// TwinCAT 3 PLC project Main_Lube_oil_Temperature_Simulation
// ProgramVersion: 3.1.4024.0
// libraries:
//   Tc2_Standard, * (Beckhoff Automation GmbH)
//   Tc2_System, * (Beckhoff Automation GmbH)
//   Tc3_Module, * (Beckhoff Automation GmbH)
//   Tc2_ControllerToolbox,3.4.3.0,Beckhoff Automation GmbH
// project tree:
//   GVLs/ MainLubeOil_Parameters.TcGVL, Simulation_Parameters.TcGVL
//   / PlcTask.TcTTO
//   POUs/ FB_RampGeneration.TcPOU, FB_ReservoirVolume.TcPOU, FB_PumpFlow.TcPOU, FB_TemperatureAfterGearbox.TcPOU, FB_TemperatureAfterPump.TcPOU, FB_TemperatureAfterHeatExchanger.TcPOU, F_Scale.TcPOU, MAIN.TcPOU, f_CalculateDeltaT.TcPOU, f_deltaT_AfterMixingTwoFluids.TcPOU, FB_ReservoirTemperature.TcPOU, FB_ReservoirHeaterIsOn.TcPOU, f_ReservoirConvectionHeat.TcPOU
// real-time tasks:
//   TASK PlcTask: cycle T#10ms, priority 20, ADS port 350

CONFIGURATION Main_Lube_oil_Temperature_Simulation
    RESOURCE PLC ON TwinCAT3
        TASK PlcTask(INTERVAL := T#10ms, PRIORITY := 20);
        PROGRAM MAIN WITH PlcTask : MAIN;
    END_RESOURCE
END_CONFIGURATION

// ---- GVLs/MainLubeOil_Parameters.TcGVL
{attribute 'qualified_only'}
VAR_GLOBAL CONSTANT
	MainLubeOilReservoirVolume : REAL := 900 ; //Liters
	MainLubeOilTotalPipeVolume: REAL := 150 ; //Liters
	
	MainLubeOilReservoirHeaterPower : REAL := 5000 ; //Watt
	MainLubeOilReservoirHeaterSPon :  REAL := 40 ; // Celcius
	MainLubeOilReservoirHeaterSPoff :  REAL := 50 ; // Celcius
	
	MainLubeOilHeatExchangerPower :  REAL := 50000 ; //Watt
	MainLubeOilHeatExchangerValveClosedTemp :  REAL := 40 ; //Celcius, Valve 0% no cooling
	MainLubeOilHeatExchangerValveOpenTemp :  REAL := 80 ; //Celcius Valve 100% max cooling
	
	
	MainLubeOilPumpPower  :  REAL := 5000 ; //Watt
	MainLubeOilPumpEfficiency :  REAL := 0.95 ; // % formatted as a decimal
	
	MainLubeOilGearboxHeat :  REAL := 5000000 ; // Watt
	MainLubeOilGearboxEfficiency :  REAL := 0.993 ; // % formatted as a deimal number
	MainLubeOilGearboxStandardHeat :  REAL := 1000 ; // Watt
	
END_VAR

// ---- GVLs/Simulation_Parameters.TcGVL
{attribute 'qualified_only'}
VAR_GLOBAL CONSTANT
	OilDensity : REAL := 865 ; // g/L
	SpecificHeatCapacityOil : REAL := 2 ; // j/(g C)
	
	AmbientTemperature : REAL := 15 ; //Celcius
	GravityOilFlow : REAL := 1 ; // L/s
	CycleTime : REAL := 0.010 ; // s , 10 ms

END_VAR
VAR_GLOBAL
	TimeConstantReservoir : REAL := 0.1 ;
	TimeConstantPump : REAL := 0.0001 ;
	TimeConstantHeatExchanger : REAL := 0.0001 ;
	TimeConstantGearbox : REAL := 0.0001 ;
END_VAR

// ---- POUs/MAIN.TcPOU
PROGRAM MAIN

VAR
	fb_MainLubeOilReservoirTemperature : FB_ReservoirTemperature ;
	fb_MainLubeOilReservoirHeaterIsOn : FB_ReservoirHeaterIsOn ;
	fb_MainLubeOilTemperatureAfterPump : FB_TemperatureAfterPump ;
	fb_MainLubeOilTemperatureAfterHeatExchanger : FB_TemperatureAfterHeatExchanger ;
	fb_MainLubeOilTemperatureAfterGearbox : FB_TemperatureAfterGearbox ;
	fb_MainLubeOilReservoirVolume : FB_ReservoirVolume ;
	fb_MainLubeOilPumpFlow : FB_PumpFlow ;
	
	MainLubeOilReservoirTemperature : REAL := simulation_parameters.AmbientTemperature; // Celcius
	MainLubeOilTemperatureAfterPump : REAL := simulation_parameters.AmbientTemperature ; // Celcius
	MainLubeOilTemperatureAfterHeatExchanger : REAL := simulation_parameters.AmbientTemperature ; // Celcius
	MainLubeOilTemperatureAfterGearbox : REAL :=simulation_parameters.AmbientTemperature ; // Celcius

	MainLubeOilReservoirVolume : REAL := MainLubeOil_Parameters.MainLubeOilReservoirVolume; // L
	MainLubeOilPumpFlow  :  REAL := 0 ; // L/s
	MainLubeOilCurrentPipeVolume : REAL := 0 ; //L

	BoolSimulationTesting : BOOL := FALSE ;
	MainLubeOilReservoirHeaterIsOn : BOOL ;
	MainLubeOilPumpOneOn : BOOL := FALSE ;
	MainLubeOilPumpTwoOn : BOOL := FALSE ;
END_VAR

fb_MainLubeOilReservoirVolume(	ReservoirVolume := MainLubeOilReservoirVolume,
								ReservoirStartVolume := MainLubeOil_Parameters.MainLubeOilReservoirVolume,
								TotalPipeVolume := MainLubeOil_Parameters.MainLubeOilTotalPipeVolume,
								PumpFlow := MainLubeOilPumpFlow);

fb_MainLubeOilPumpFlow(	PumpOneOn := MainLubeOilPumpOneOn, 
						PumpTwoOn := MainLubeOilPumpTwoOn) ;
	
fb_MainLubeOilReservoirTemperature(	ReservoirVolume := MainLubeOilReservoirVolume,
									ReservoirHeaterIsOn := MainLubeOilReservoirHeaterIsOn,
									TotalPipeVolume := MainLubeOil_Parameters.MainLubeOilTotalPipeVolume,
									CurrentPipeVolume := MainLubeOilCurrentPipeVolume,
									TemperatureAfterGearbox := MainLubeOilTemperatureAfterGearbox);

									
fb_MainLubeOilReservoirHeaterIsOn(ReservoirTemperature := MainLubeOilReservoirTemperature,
								ReservoirHeaterIsOn := MainLubeOilReservoirHeaterIsOn,
								ReservoirHeaterSPon := MainLubeOil_Parameters.MainLubeOilReservoirHeaterSPon,
								ReservoirHeaterSPoff := MainLubeOil_Parameters.MainLubeOilReservoirHeaterSPoff,
								BoolSimulationTesting := BoolSimulationTesting);
								
fb_MainLubeOilTemperatureAfterPump(	TemperatureBeforePump := MainLubeOilReservoirTemperature, 
									PumpPower := MainLubeOil_Parameters.MainLubeOilPumpPower,
									PumpFlow := MainLubeOilPumpFlow,
									Density := simulation_parameters.OilDensity,
									SpecificHeatCapacity := simulation_parameters.SpecificHeatCapacityOil,
									PumpEfficiency := MainLubeOil_Parameters.MainLubeOilPumpEfficiency)	;				

fb_MainLubeOilTemperatureAfterHeatExchanger(TemperatureBeforeHeatExchanger:= MainLubeOilTemperatureAfterPump,
											HeatExchangerPower := MainLubeOil_Parameters.MainLubeOilHeatExchangerPower ,
											PumpFlow := MainLubeOilPumpFlow,
											Density := Simulation_Parameters.OilDensity,
											SpecificHeatCapacity := Simulation_Parameters.SpecificHeatCapacityOil,
											Heatexchangervalveclosedtemp :=MainLubeOil_Parameters.MainLubeOilHeatExchangerValveClosedTemp ,
											HeatExchangerValveOpenTemp := MainLubeOil_Parameters.MainLubeOilHeatExchangerValveOpenTemp,
											TotalPipeVolume := MainLubeOil_Parameters.MainLubeOilTotalPipeVolume,
											CurrentPipeVolume := MainLubeOilCurrentPipeVolume,
											BoolSimulationTesting := BoolSimulationTesting);

fb_MainLubeOilTemperatureAfterGearbox(	TemperatureBeforeGearbox:= MainLubeOilTemperatureAfterHeatexchanger,
										PumpFlow := MainLubeOilPumpFlow,
										Density := Simulation_Parameters.OilDensity,
										SpecificHeatCapacity := Simulation_Parameters.SpecificHeatCapacityOil,
										GearboxEfficiency := MainLubeOil_Parameters.MainLubeOilGearboxEfficiency,
										Gearboxheat := MainLubeOil_Parameters.MainLubeOilGearboxHeat,
										GearboxStandardHeat := MainLubeOil_Parameters.MainLubeOilGearboxStandardHeat,
										TotalPipeVolume := MainLubeOil_Parameters.MainLubeOilTotalPipeVolume,
										CurrentPipeVolume := MainLubeOilCurrentPipeVolume,
										BoolSimulationTesting := BoolSimulationTesting);								
								
MainLubeOilReservoirTemperature := fb_MainLubeOilReservoirTemperature.ReservoirTemperature ;
MainLubeOilReservoirHeaterIsOn := fb_MainLubeOilReservoirHeaterIsOn.ReservoirHeaterIsOn ;
MainLubeOilTemperatureAfterPump := fb_MainLubeOilTemperatureAfterPump.TemperatureAfterPump ;
MainLubeOilTemperatureAfterHeatExchanger := fb_MainLubeOilTemperatureAfterHeatExchanger.TemperatureAfterHeatexchanger ;
MainLubeOilTemperatureAfterGearbox := fb_MainLubeOilTemperatureAfterGearbox.TemperatureAfterGearbox ;
MainLubeOilReservoirVolume := fb_MainLubeOilReservoirVolume.ReservoirVolume ;
MainLubeOilCurrentPipeVolume := fb_MainLubeOilReservoirVolume.CurrentPipeVolume ;
MainLubeOilPumpFlow := fb_MainLubeOilPumpFlow.PumpFlow ;

END_PROGRAM

// ---- POUs/FB_ReservoirTemperature.TcPOU
FUNCTION_BLOCK FB_ReservoirTemperature
VAR_INPUT
	ReservoirVolume : REAL ; // L
	ReservoirHeaterIsOn : BOOL ;
	TotalPipeVolume : REAL ; // L
	CurrentPipeVolume : REAL ; // L
	TemperatureAfterGearbox : REAL ; //Celcius
END_VAR
VAR_OUTPUT
	ReservoirTemperature : REAL := Simulation_Parameters.AmbientTemperature ; //Celcius
END_VAR
VAR
	deltaTHeater : REAL := 0; // Celcius
	deltaTMixingGearboxReturn : REAL :=0 ; // Celcius
	
	ReservoirTemperatureNonFiltered : REAL := Simulation_Parameters.AmbientTemperature; // Celcius
	ReservoirConvectionHeat : REAL := 0 ; // Watt
	deltaTConvection : REAL := 0; // Celcius
	AmbientTemperature : REAL := Simulation_Parameters.AmbientTemperature; // Celcius
END_VAR

IF CurrentPipeVolume < (TotalPipeVolume) THEN
	deltaTMixingGearboxReturn := 0 ;
ELSE
	deltaTMixingGearboxReturn := f_deltaT_AfterMixingTwoFluids(	Mass1 := main.fb_MainLubeOilTemperatureAfterGearbox.PumpFlow,
																						SpecificHeatCapacity1 := simulation_parameters.SpecificHeatCapacityOil,
																						Temperature1 := TemperatureAfterGearbox,
																						Mass2 := ReservoirVolume,
																						SpecificHeatCapacity2 := simulation_parameters.SpecificHeatCapacityOil,
																						Temperature2 := ReservoirTemperature);
END_IF

	

IF ReservoirHeaterIsOn THEN
	deltaTHeater := f_CalculateDeltaT(	SpecificHeatCapacity := simulation_parameters.SpecificHeatCapacityOil,
										Density := Simulation_Parameters.OilDensity,
										Mass := ReservoirVolume,
										PowerInput := MainLubeoil_parameters.MainLubeOilReservoirHeaterPower);
ELSIF NOT ReservoirHeaterIsOn  THEN
	deltaTHeater := 0;
END_IF

ReservoirConvectionHeat := f_ReservoirConvectionHeat(ReservoirTemperature := ReservoirTemperature,
														AmbientTemperature := AmbientTemperature) ;
deltaTConvection := f_CalculateDeltaT (	SpecificHeatCapacity := simulation_parameters.SpecificHeatCapacityOil,
										Density := Simulation_Parameters.OilDensity,
										Mass := ReservoirVolume,
										PowerInput := ReservoirConvectionHeat);
										
ReservoirTemperatureNonFiltered := ReservoirTemperature + deltaTHeater + deltaTMixingGearboxReturn - deltaTConvection;
ReservoirTemperature := (1-simulation_parameters.TimeConstantReservoir)*ReservoirTemperature + simulation_parameters.TimeConstantReservoir*ReservoirTemperatureNonFiltered ;

END_FUNCTION_BLOCK

// ---- POUs/f_deltaT_AfterMixingTwoFluids.TcPOU
FUNCTION f_deltaT_AfterMixingTwoFluids : REAL
VAR_INPUT
	Mass1 : REAL ; // g
	SpecificHeatCapacity1 : REAL ; //  j/(g C), 
	Temperature1 : REAL ; // Celcius
	
	Mass2 : REAL ; // g
	SpecificHeatCapacity2 : REAL ; //  j/(g C), 
	Temperature2 : REAL ; // Celcius
END_VAR

f_deltaT_AfterMixingTwoFluids := ((Mass1 * SpecificHeatCapacity1 * Temperature1)+(Mass2 * SpecificHeatCapacity2 * Temperature2))/((Mass1 * SpecificHeatCapacity1 )+(Mass2 * SpecificHeatCapacity2 )) - Temperature2;

END_FUNCTION

// ---- POUs/f_CalculateDeltaT.TcPOU
FUNCTION f_CalculateDeltaT : REAL

VAR_INPUT
	PowerInput : REAL ; // Watts
	Density : REAL ; // g/L
	SpecificHeatCapacity : REAL ; // j/(g C)
	Mass : REAL; // g
END_VAR

IF Density =0 OR SpecificHeatCapacity =0 OR Mass =0 THEN 
	f_CalculateDeltaT := 0 ; 
ELSIF Mass < 0.3 THEN  //Filter to prevent large spikes when dividing by very small mass numbers.
	f_CalculateDeltaT := 0 ; 
ELSE
	f_CalculateDeltaT := PowerInput / (Density * SpecificHeatCapacity * Mass);
END_IF

END_FUNCTION

// ---- POUs/f_ReservoirConvectionHeat.TcPOU
FUNCTION f_ReservoirConvectionHeat : REAL
VAR_INPUT
	ReservoirTemperature : REAL ; // Celcius
	AmbientTemperature : REAL ; // Celcius
END_VAR
VAR_OUTPUT
	ReservoirConvectionHeat: REAL ; // Watt
END_VAR
VAR
	ConvectiveHeatTransferCoeff : REAL := 10 ; // Watt/(m2 K)
	ReservoirSurfaceArea : REAL :=6 ; // m2
END_VAR

f_ReservoirConvectionHeat := ConvectiveHeatTransferCoeff * ReservoirSurfaceArea * (ReservoirTemperature - AmbientTemperature);

END_FUNCTION

// ---- POUs/FB_ReservoirHeaterIsOn.TcPOU
FUNCTION_BLOCK FB_ReservoirHeaterIsOn
VAR_INPUT
	ReservoirTemperature : REAL ; // Celcius
	ReservoirHeaterIsOn : BOOL ; 
	ReservoirHeaterSPon : REAL ; // Celcius
	ReservoirHeaterSPoff : REAL ; // Celcius
	BoolSimulationTesting : BOOL ; //True if testing with PLC logic
END_VAR

IF NOT BoolSimulationTesting THEN
	IF (ReservoirTemperature < ReservoirHeaterSPon) THEN
		ReservoirHeaterIsOn := TRUE ; 
	ELSIF ((ReservoirTemperature > ReservoirHeaterSPon) AND (ReservoirTemperature < ReservoirHeaterSPoff)) AND ReservoirHeaterIsOn THEN
		ReservoirHeaterIsOn :=TRUE; 
	ELSIF ((ReservoirTemperature > ReservoirHeaterSPon) AND (ReservoirTemperature < ReservoirHeaterSPoff)) AND NOT ReservoirHeaterIsOn THEN
		ReservoirHeaterIsOn :=FALSE;
	ELSIF (ReservoirTemperature > ReservoirHeaterSPoff) THEN
		ReservoirHeaterIsOn :=FALSE;
	END_IF
END_IF

END_FUNCTION_BLOCK

// ---- POUs/FB_TemperatureAfterPump.TcPOU
FUNCTION_BLOCK FB_TemperatureAfterPump
VAR_INPUT
	TemperatureBeforePump : REAL ; // Celcius
	PumpPower : REAL ; // Watt
	PumpFlow : REAL ; // L/s
	Density : REAL ; // g/L
	SpecificHeatCapacity : REAL ; //  j/(g C)
	PumpEfficiency : REAL ; //% 0-1
END_VAR
VAR_OUTPUT
	TemperatureAfterPump : REAL := Simulation_Parameters.AmbientTemperature ; // Celcius
END_VAR
VAR
	deltaTByPump : REAL ; // Celcius
	TemperatureAfterPumpNonFiltered : REAL ; //Celcius
END_VAR

IF PumpFlow = 0 THEN
	;
ELSE
	deltaTByPump := f_CalculateDeltaT(	SpecificHeatCapacity := SpecificHeatCapacity,
									Density := Density,
									Mass := PumpFlow,
									PowerInput := PumpPower);
					
	TemperatureAfterPumpNonFiltered := TemperatureBeforePump + ( (1 - PumpEfficiency) * deltaTByPump ) ;	
	TemperatureAfterPump := (1-simulation_parameters.TimeConstantPump)*TemperatureAfterPump + simulation_parameters.TimeConstantPump*TemperatureAfterPumpNonFiltered ;
END_IF

END_FUNCTION_BLOCK

// ---- POUs/FB_TemperatureAfterHeatExchanger.TcPOU
FUNCTION_BLOCK FB_TemperatureAfterHeatExchanger
VAR_INPUT
	TemperatureBeforeHeatExchanger : REAL ; // Celsius
	HeatExchangerPower : REAL ; // Watt
	PumpFlow : REAL ; // L/s
	Density : REAL ; // g/L
	SpecificHeatCapacity : REAL ; // j/(g C)
	
	HeatExchangerValveClosedTemp : REAL ; // Celsius
	HeatExchangerValveOpenTemp : REAL ; // Celsius
	TotalPipeVolume : REAL ; // L
	CurrentPipeVolume : REAL ; // L
	BoolSimulationTesting : BOOL ;
END_VAR
VAR_OUTPUT
	TemperatureAfterHeatExchanger : REAL := Simulation_Parameters.AmbientTemperature; // Celcius
END_VAR
VAR
	HeatExchangerValvePercentageOpen : REAL ; //% 0-1
	HeatExchangerValveMaxOpen : REAL := 1; //1 = 100%
	HeatExchangerValveMinOpen : REAL := 0; //0 = 0%
	deltaTByHeatExchanger : REAL ; // Celcius
	
	MimimumPipeVolumeForHeatTransfer : REAL ; // L
	TemperatureAfterHeatExchangerNonFiltered : REAL ; // Celcius
END_VAR

IF NOT BoolSimulationTesting THEN
	IF TemperatureBeforeHeatExchanger < HeatExchangerValveClosedTemp THEN
		HeatExchangerValvePercentageOpen :=0 ;
	ELSIF TemperatureBeforeHeatExchanger > HeatExchangerValveOpenTemp THEN
		HeatExchangerValvePercentageOpen :=100 ;
	ELSE 
		HeatExchangerValvePercentageOpen := F_Scale(inputValue :=TemperatureBeforeHeatExchanger,
													inputMaxValue := HeatExchangerValveOpenTemp,
													InputMinValue := HeatExchangerValveClosedTemp,
													inputScaleMaxLimit := HeatExchangerValveMaxOpen,
													inputScaleMinLimit := HeatExchangerValveMinOpen);
	END_IF
ELSE
	//HeatExchangerValvePercentageOpen value of PLC simulation
END_IF

MimimumPipeVolumeForHeatTransfer := TotalPipeVolume/4;
IF CurrentPipeVolume <= MimimumPipeVolumeForHeatTransfer THEN
	deltaTByHeatExchanger := 0 ;
ELSE 
	deltaTByHeatExchanger := f_CalculateDeltaT(SpecificHeatCapacity := SpecificHeatCapacity,
												Density := Density,
												Mass := PumpFlow,
												PowerInput := HeatExchangerPower);
								
	TemperatureAfterHeatExchangerNonFiltered := TemperatureBeforeHeatExchanger - ( (HeatExchangerValvePercentageOpen) * deltaTByHeatExchanger ) ;
	TemperatureAfterHeatExchanger := (1-simulation_parameters.TimeConstantHeatExchanger)*TemperatureAfterHeatExchanger + simulation_parameters.TimeConstantHeatExchanger*TemperatureAfterHeatExchangerNonFiltered ;
END_IF

END_FUNCTION_BLOCK

// ---- POUs/F_Scale.TcPOU
FUNCTION F_Scale : REAL

VAR_INPUT
	inputValue : REAL;
	inputMaxValue : REAL;
	inputMinValue : REAL;
	inputScaleMaxLimit : REAL; 
	inputScaleMinLimit : REAL;
END_VAR

VAR
	fNormalizedValue : REAL :=0;
	fScaledValue : REAL := 0;
END_VAR

//Normalize the  input
IF inputValue < inputMinValue THEN
	fNormalizedValue := 0;
ELSIF inputValue > 	inputMaxValue THEN
	fNormalizedValue := 1;
ELSE
	fNormalizedValue := (inputValue - inputMinValue) / (inputMaxValue - inputMinValue);
END_IF

//Scale the output
F_Scale := fNormalizedValue * (inputScaleMaxLimit - inputScaleMinLimit) + inputScaleMinLimit;

END_FUNCTION

// ---- POUs/FB_TemperatureAfterGearbox.TcPOU
FUNCTION_BLOCK FB_TemperatureAfterGearbox
VAR_INPUT
	TemperatureBeforeGearbox : REAL ; // Celcius
	PumpFlow : REAL ; // L/s
	Density : REAL ; // g/L
	SpecificHeatCapacity : REAL ; //  j/(g C) 
	GearboxEfficiency : REAL ; //%, 0-1
	Gearboxheat : REAL ; // Watt
	GearboxStandardHeat : REAL ; // Watt
	TotalPipeVolume : REAL ; // L
	CurrentPipeVolume : REAL ; // L
	BoolSimulationTesting : BOOL ;
END_VAR
VAR_OUTPUT
	TemperatureAfterGearbox : REAL := Simulation_Parameters.AmbientTemperature ; // L
END_VAR
VAR
	SurgeValvePosition : REAL ; // % 0-1
	deltaTByGearboxHeat : REAL ; // Celsius
	deltaTByGearboxStandardHeat : REAL ; // Celsius
	deltaTByGearboxHeatEfficiencyCorrected : REAL ; // Celsius
	
	MimimumPipeVolumeForHeatTransfer : REAL ; // L
	TemperatureAfterGearboxNonFiltered : REAL ; // Celsius
END_VAR

IF NOT BoolSimulationTesting THEN
	SurgeValvePosition := 0.05; //Use hardcoded SurgeValvePosition
ELSE
	; //Frank Logic for SurgeValvePosition.
END_IF


MimimumPipeVolumeForHeatTransfer := TotalPipeVolume*3/4;

IF CurrentPipeVolume <= MimimumPipeVolumeForHeatTransfer THEN
	deltaTByGearboxHeat := 0 ;
	deltaTByGearboxStandardHeat := 0 ;
	
ELSE 
	deltaTByGearboxHeat := f_CalculateDeltaT(SpecificHeatCapacity := SpecificHeatCapacity,
											Density := Density,
											Mass := PumpFlow,
											PowerInput := Gearboxheat);
								
	deltaTByGearboxStandardHeat := f_CalculateDeltaT(SpecificHeatCapacity := SpecificHeatCapacity,
													Density := Density,
													Mass := PumpFlow,
													PowerInput := GearboxStandardHeat); 
	deltaTByGearboxHeatEfficiencyCorrected := (1-GearboxEfficiency) * deltaTByGearboxHeat;
						
	TemperatureAfterGearboxNonFiltered := TemperatureBeforeGearbox + (SurgeValvePosition *  deltaTByGearboxHeatEfficiencyCorrected) + deltaTByGearboxStandardHeat;
	TemperatureAfterGearbox := (1-simulation_parameters.TimeConstantGearbox)*TemperatureAfterGearbox + simulation_parameters.TimeConstantGearbox*TemperatureAfterGearboxNonFiltered ;

END_IF

END_FUNCTION_BLOCK

// ---- POUs/FB_ReservoirVolume.TcPOU
FUNCTION_BLOCK FB_ReservoirVolume
VAR_INPUT
	ReservoirVolume : REAL; // L
	ReservoirStartVolume : REAL ; // L
	TotalPipeVolume : REAL ; // L
	PumpFlow : REAL ; // L/s
	
END_VAR
VAR_OUTPUT
	CurrentPipeVolume : REAL ;
END_VAR
VAR
END_VAR

IF (ReservoirVolume <= ReservoirStartVolume) AND (ReservoirVolume >=(ReservoirStartVolume - TotalPipeVolume) ) THEN
	ReservoirVolume := ReservoirVolume - PumpFlow / (1/simulation_parameters.CycleTime) + simulation_parameters.GravityOilFlow/(1/simulation_parameters.CycleTime) ;
	IF ReservoirVolume > ReservoirStartVolume THEN
		ReservoirVolume :=ReservoirStartVolume ;
	ELSIF (ReservoirVolume <= (ReservoirStartVolume - TotalPipeVolume)) THEN
		ReservoirVolume := (ReservoirStartVolume - TotalPipeVolume) ;
	END_IF
ELSIF (ReservoirVolume >= ReservoirStartVolume) THEN
	ReservoirVolume := ReservoirStartVolume - PumpFlow / (1/simulation_parameters.CycleTime);
ELSIF (ReservoirVolume <= (ReservoirStartVolume - TotalPipeVolume)) THEN
	ReservoirVolume := (ReservoirStartVolume - TotalPipeVolume) + simulation_parameters.GravityOilFlow/(1/simulation_parameters.CycleTime) ;
END_IF

IF ReservoirVolume <= ReservoirStartVolume THEN
	CurrentPipeVolume := ReservoirStartVolume - ReservoirVolume ;
END_IF

END_FUNCTION_BLOCK

// ---- POUs/FB_PumpFlow.TcPOU
FUNCTION_BLOCK FB_PumpFlow
VAR_INPUT
	PumpOneOn : BOOL;
	PumpTwoOn : BOOL ;
	PumpFlow : REAL ; // L/s
END_VAR
VAR
	fb_ramp_generation : FB_RampGeneration ;
	PumpFlowTarget : REAL := 0; // L/s
	RampTimeStepPumpFlow : REAL :=0.1; //100ms call
	RampFactorPumpFlow : REAL :=0.3; // Velocity ramp
END_VAR

IF (PumpOneOn AND PumpTwoOn) THEN
	PumpFlowTarget := 6 ;

ELSIF (PumpOneOn OR PumpTwoOn)  THEN
	PumpFlowTarget :=3 ;
ELSIF NOT (PumpOneOn AND PumpTwoOn)  THEN
	PumpFlowTarget :=0;
END_IF

fb_ramp_generation(RampStart :=PumpFlow, 
					RampTarget := PumpFlowTarget, 
					RampTimestep := RampTimeStepPumpFlow, 
					RampFactor := RampFactorPumpFlow) ;
pumpflow := fb_ramp_generation.RampOutput ;

END_FUNCTION_BLOCK

// ---- POUs/FB_RampGeneration.TcPOU
FUNCTION_BLOCK FB_RampGeneration
VAR_INPUT
RampStart : REAL ; //Start value of ramp
RampTarget : REAL ; //Target Value of ramp
RampTimeStep : REAL ; //100ms call
RampFactor : REAL ; //Units added
END_VAR

VAR_OUTPUT
RampOutput : REAL ;
END_VAR

IF RampStart < RampTarget THEN
	RampStart := RampStart + (RampFactor * RampTimeStep) ;
	IF (RampStart > RampTarget) THEN
		RampStart := RampTarget ;
	END_IF
END_IF 

IF RampStart > RampTarget THEN  
	RampStart := RampStart - (RampFactor * RampTimeStep) ;
	IF (RampStart < RampTarget) THEN
		RampStart := RampTarget;
	END_IF
END_IF

RampOutput := RampStart ;

END_FUNCTION_BLOCK
